FUNCTION_BLOCK StationSequence IMPLEMENTS I_Cyclic, I_Resettable, I_Object
VAR
	State : StationSequenceState;  
	CurrentStation : UINT;
	TargetStationPosition : MC_LREAL;
	_MoverVelocity : MC_LREAL := 1000.0;
	stSequenceInfo : SequenceInfo;
	StationNumber : INT;
	StationArray : ARRAY[0..19] OF IStation;
	Process : IProcess;
	ThisMover : I_XtsMover;
	ExecuteSequence : BOOL;
	_startPosition : MC_LREAL;
	_XtsNoHome : BOOL;
	_NonModuloMoves : BOOL := FALSE;
END_VAR

{analysis -2}

METHOD PUBLIC Cycle : HRESULT
VAR_INPUT
END_VAR
CASE State OF
	StationSequenceState.Init:
		IF ThisMover.isMoverEnabled() THEN
			State := StationSequenceState.Available;
		END_IF
		
	StationSequenceState.Available:
		IF ExecuteSequence THEN
			State := StationSequenceState.MovingToStart;
		END_IF
		
	StationSequenceState.MovingToStart:
		IF ThisMover.isMoverAtPosition(position := _startPosition) OR _XtsNoHome THEN
			State := StationSequenceState.AtStart;
		END_IF
			
	StationSequenceState.AtStart:
		IF StationArray[CurrentStation] <> 0 AND_THEN StationArray[CurrentStation].IsReady() THEN
			IF SUCCEEDED(ThisMover.MoveTo(RequiredPosition := StationArray[CurrentStation].Position,
								MoveVelocity := _MoverVelocity,
								NonModuloMove := _NonModuloMoves)) THEN
								
				TargetStationPosition := StationArray[CurrentStation].Position;
				State := StationSequenceState.MovingToStation;
			END_IF
		END_IF

	StationSequenceState.MovingToStation:
		IF ThisMover.isMoverStationary() THEN 
			IF ThisMover.isMoverAtPosition(TargetStationPosition) THEN
				IF __QUERYINTERFACE(StationArray[CurrentStation],Process) THEN
					State := StationSequenceState.AtProcess;
				ELSE
					State := StationSequenceState.AtStation;
				END_IF
				StationArray[CurrentStation].MyMover(ThisMover);
			ELSE
				State := StationSequenceState.QueuedAtStation;
			END_IF
		END_IF
		
	StationSequenceState.QueuedAtStation:
		IF NOT ThisMover.isMoverStationary() THEN
				State := StationSequenceState.MovingToStation;
		END_IF

	StationSequenceState.AtStation:
		IF StationArray[CurrentStation].isComplete() THEN
			State := StationSequenceState.GetNextMove;
		END_IF

	StationSequenceState.AtProcess:
		ThisMover.MoveTo(RequiredPosition := Process.EndPosition,
								MoveVelocity := Process.ProcessVelocity,
								NonModuloMove := _NonModuloMoves);
		State := StationSequenceState.InProcess;
								
	StationSequenceState.InProcess:
		IF ThisMover.isMoverStationary() THEN 
			IF ThisMover.isMoverAtPosition(Process.EndPosition) THEN
				State := StationSequenceState.GetNextMove;
			END_IF
		END_IF
	
	StationSequenceState.GetNextMove:
		IF CurrentStation = StationNumber - 1 THEN
			CurrentStation := 0; 
			IF SUCCEEDED(ThisMover.MoveTo(RequiredPosition := StationArray[CurrentStation].Position,
							MoveVelocity := _MoverVelocity,
							NonModuloMove := _NonModuloMoves)) THEN
				State := StationSequenceState.MovingToStation;
				TargetStationPosition := StationArray[CurrentStation].Position;
			END_IF
		ELSE
			State := StationSequenceState.GoToNextStation;
		END_IF
		
	StationSequenceState.GoToNextStation:
		TargetStationPosition := StationArray[CurrentStation + 1].Position;
		IF 	SUCCEEDED(ThisMover.MoveTo(RequiredPosition := TargetStationPosition,
							MoveVelocity := _MoverVelocity,
							NonModuloMove := _NonModuloMoves)) THEN	
			CurrentStation := CurrentStation + 1;
			State := StationSequenceState.MovingToStation;
		END_IF	

	StationSequenceState.Stopping:
		State := StationSequenceState.Available;
		CurrentStation := 0;
		TargetStationPosition := 0.0;
	ELSE
		Cycle := E_FAIL;
END_CASE

//Cyclic update info data
stSequenceInfo.CurrentStation := UINT_TO_INT(CurrentStation);
stSequenceInfo.MoverId := ThisMover.AxisRef.NcToPlc.AxisId;
stSequenceInfo.State := State;
stSequenceInfo.Velocity := ThisMover.AxisRef.NcToPlc.ActVelo;
END_METHOD

PROPERTY MoverVelocity : mc_lreal
GET
MoverVelocity := _MoverVelocity;
END_GET
SET
_MoverVelocity := MoverVelocity;
END_SET
END_PROPERTY

PROPERTY MyMover : I_XtsMover
GET
MyMover := ThisMover;
END_GET
SET
ThisMover := MyMover;
END_SET
END_PROPERTY

PROPERTY MyStartPosition : MC_LREAL
GET
MyStartPosition := _startPosition;
END_GET
SET
_startPosition := MyStartPosition;
END_SET
END_PROPERTY

METHOD RegisterAStation : HRESULT
VAR_INPUT
	Station : IStation;
END_VAR
IF Station = 0 THEN
	RegisterAStation  := -1;
	RETURN;
END_IF
StationArray[StationNumber] := Station;
StationNumber := StationNumber + 1;
END_METHOD

METHOD RegisterWithParent
VAR_INPUT
	Runner	: I_HostObjects;
END_VAR
Runner.RegisterCyclic(THIS^);
END_METHOD

METHOD Reset : HRESULT
VAR_INPUT
END_VAR
State := StationSequenceState.Available;
CurrentStation := 0;
TargetStationPosition := 0.0;
stSequenceInfo.CurrentStation := UINT_TO_INT(CurrentStation);
stSequenceInfo.MoverId := ThisMover.AxisRef.NcToPlc.AxisId;
stSequenceInfo.State := State;
stSequenceInfo.Velocity := ThisMover.AxisRef.NcToPlc.ActVelo;
ExecuteSequence := FALSE;
Reset := 1;
END_METHOD

METHOD StartIndexing : BOOL
VAR_INPUT
END_VAR
ExecuteSequence := TRUE;
END_METHOD

PROPERTY XtsNoHome : BOOL
GET
XtsNoHome := _XtsNoHome;
END_GET
SET
_XtsNoHome := XtsNoHome;
END_SET
END_PROPERTY

END_FUNCTION_BLOCK

(* stored: Version 1.1.0.1
   POU StationSequence: Id {50af290e-a0d7-45b3-a647-c8828b096bd1}, SpecialFunc None
   Method Cycle: Id {0bc270b2-0e7a-4545-b872-87f2d15ca3f5}
   Property MoverVelocity: Id {4f2224ad-0534-4bd9-a8e4-5b63b7e53b5c}
   Get Get: Id {0bf3cfa6-cc44-4232-989f-70bced017a55}
   Set Set: Id {a9bdfb5a-ef56-4b9e-9f78-288684e24d6c}
   Property MyMover: Id {d0dbd650-93c6-4e7f-a733-abc40a2f12bf}
   Get Get: Id {52e46adf-1b9f-404f-a8d7-de686d91d4ef}
   Set Set: Id {a9693a81-065c-4ba2-8a99-3606c71cf06a}
   Property MyStartPosition: Id {30ed087d-d896-49f8-aaff-c511c0d55a71}
   Get Get: Id {ebcb0d89-302c-4f5d-86e5-f5e15f136ea5}
   Set Set: Id {57b76837-f6ca-44d6-8033-7a2d9ee3e944}
   Method RegisterAStation: Id {14d9a1a8-6162-46e7-9803-61945cdf77e8}
   Method RegisterWithParent: Id {4ad7e011-f71b-4cbe-b657-57f840858ed2}
   Method Reset: Id {01dd3306-e903-4754-85c4-ea13c41e0b8c}
   Method StartIndexing: Id {6e4b7f28-1f53-404c-b56b-f1310c888415}
   Property XtsNoHome: Id {7aad9af3-71dc-4b8d-9a2b-19016c2a644b}
   Get Get: Id {d3413585-01ef-4909-a612-e4cda3a7b8e0}
   Set Set: Id {ca6f67d3-9265-4c0f-849c-5e4c98f82e9b} *)
